(* CODESYS project PlcLibrary1_1.2.3.3.library
   Title: PlcLibrary1
   Version: 1.2.3.3
   Placeholder: PlcLibrary1
   Company: My Company

Project tree, tasks and I/O mapping:
  libraries: Tc2_Standard, * (Beckhoff Automation GmbH); Tc2_System, * (Beckhoff Automation GmbH)
  DUTs/
  GVLs/
  POUs/
    program MAIN [ST]
  VISUs/
*)

// POUs/MAIN
PROGRAM MAIN
VAR
END_VAR

END_PROGRAM
